SUBAPPLICATION Uebung_042 (* Scaling Function Block Testing *)
  (* Standard: 61499-2 *)
  (* Version 1.0, 2023-10-23, franz *)
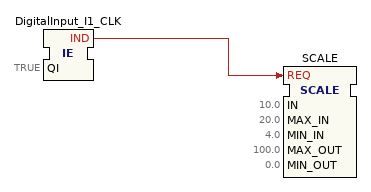
  FBS
    DigitalInput_I1_CLK : IE(QI := TRUE);
    SCALE : signalprocessing::SCALE(IN := 10.0, MAX_IN := 20.0, MIN_IN := 4.0, MAX_OUT := 100.0, MIN_OUT := 0.0);
  END_FBS
  EVENT_CONNECTIONS
    DigitalInput_I1_CLK.IND TO SCALE.REQ;
  END_CONNECTIONS
END_SUBAPPLICATION
